FUNCTION_BLOCK QW (* Composite Function Block Type *)
  (* Standard: 61499-2 *)
  (* Version 0.0, 2016-04-07, 4DIAC-IDE, 4DIAC-Consortium *)
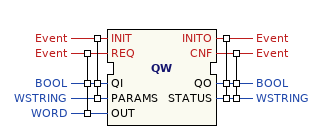
  EVENT_INPUT
    INIT WITH QI, PARAMS; (* Initialization Request *)
    REQ WITH QI, OUT; (* Normal Execution Request *)
  END_EVENT
  EVENT_OUTPUT
    INITO WITH QO, STATUS; (* Initialization Confirm *)
    CNF WITH QO, STATUS; (* Execution Confirmation *)
  END_EVENT
  VAR_INPUT
    QI : BOOL; (* Input event qualifier *)
    PARAMS : WSTRING;
    OUT : WORD;
  END_VAR
  VAR_OUTPUT
    QO : BOOL; (* Output event qualifier *)
    STATUS : WSTRING;
  END_VAR
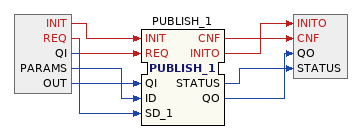
  FBS
    PUBLISH_1 : PUBLISH_1;
  END_FBS
  EVENT_CONNECTIONS
    INIT TO PUBLISH_1.INIT;
    REQ TO PUBLISH_1.REQ;
    PUBLISH_1.CNF TO CNF;
    PUBLISH_1.INITO TO INITO;
  END_CONNECTIONS
  DATA_CONNECTIONS
    QI TO PUBLISH_1.QI;
    PARAMS TO PUBLISH_1.ID;
    OUT TO PUBLISH_1.SD_1;
    PUBLISH_1.STATUS TO STATUS;
    PUBLISH_1.QO TO QO;
  END_CONNECTIONS
END_FUNCTION_BLOCK
